{attribute 'linkalways'} 
{attribute 'no_explicit_call' := 'This FB is a CLASS and must be accessed using methods or properties'}
{attribute 'enable_dynamic_creation'}
FUNCTION_BLOCK FINAL LE_UINT EXTENDS Node
VAR
	in1 : _UINT(0);
	in2 : _UINT(0);
	out : _BOOL(FALSE);
END_VAR

METHOD PUBLIC Clone : I_Node
VAR
	pNode : POINTER TO LE_UINT;
END_VAR
pNode := __NEW(LE_UINT);
Clone := pNode^;
END_METHOD

METHOD FB_init : BOOL
VAR_INPUT
	bInitRetains : BOOL; // if TRUE, the retain variables are initialized (warm start / cold start)
	bInCopyCode : BOOL;  // if TRUE, the instance afterwards gets moved into the copy code (online change)
END_VAR
AddInput('in1',THIS^.in1);
AddInput('in2',THIS^.in2);
AddOutput('out', THIS^.out);
END_METHOD

METHOD PROTECTED OnExecute
VAR
END_VAR
out.Value := in1.Value <= in2.Value;
END_METHOD

END_FUNCTION_BLOCK

(* stored: Version 1.1.0.1, ProductVersion 3.1.4024.15
   POU LE_UINT: Id {a7463258-b46e-4fc5-b349-9be541cb3982}, SpecialFunc None
   Folder Constructor: Id {1ceb8616-1db0-4471-96f3-4137238769c3}
   Method Clone: Id {47b45dc2-1401-4130-9281-56d8a99df884}
   Method FB_init: Id {bbc99bb5-4418-4216-a182-a606722b4904}
   Method OnExecute: Id {8899b8b2-b028-4077-ba70-d1b0f9080572} *)
